(*			
	EVERDE sp. z o.o.
	Rafał Osajda		27.05.2025		TC 4024.66
	Metoda główna bazowania wywołuje metode przeciążaną Bazowanie_Cykl dziecka
*)
METHOD PRIVATE HomingCycleInternal : BOOL
VAR_INPUT
END_VAR
CASE THIS^.stHoming.cmdExecute.GetStep () OF
0	:
	IF (THIS^.stHoming.bWithoutHoming) THEN	//bazowanie wyłączone true
		THIS^.stHoming.bIsNeeded		:= TRUE;	//ustaw że juz jest wybazowane
		THIS^.stHoming.cmdExecute.SetStepAsFinal ();
	ELSE
		THIS^.stHoming.iElementHomingStep	:= 0;
		THIS^.stHoming.cmdExecute.SetStepINC10 ();
	END_IF
	THIS^.stHoming.bIsNeeded			:= TRUE;
	HomingCycleInternal				:= TRUE;
10	:
	IF (NOT THIS^.HomingCycle ()) THEN
		THIS^.stHoming.cmdExecute.SetStepAsFinal ();
	END_IF
	HomingCycleInternal				:= TRUE;
GVL_BaseConstans.FINISH_STEP	:
	THIS^.stHoming.bIsNeeded			:= FALSE;	//ustaw że juz jest wybazowane
	HomingCycleInternal				:= FALSE;
END_CASE
END_METHOD

(*			
	EVERDE sp. z o.o.
	Rafał Osajda		27.05.2025		TC 4024.66
	Bazowanie w toku
*)
METHOD PUBLIC HomingGetBusy : BOOL
VAR_INPUT
END_VAR
HomingGetBusy		:= THIS^.stHoming.cmdExecute.IsBusy ();
END_METHOD

(*			
	EVERDE sp. z o.o.
	Rafał Osajda		31.03.2025		TC 4024.66
	Flaga że w tej sesji pracy maszyny element został już wybazowany
*)
METHOD PUBLIC HomingGetDone : BOOL
VAR_INPUT
END_VAR
HomingGetDone	:= THIS^.stHoming.cmdExecute.IsDone ();
END_METHOD

(*			
	EVERDE sp. z o.o.
	Rafał Osajda		11.04.2025		TC 4024.66
	Zwraca czy bazowanie jest potrzebne
*)
METHOD PUBLIC HomingGetIsNeeded : BOOL
VAR_INPUT
END_VAR
HomingGetIsNeeded			:= THIS^.stHoming.bIsNeeded;
END_METHOD

(*			
	EVERDE sp. z o.o.
	Rafał Osajda		11.04.2025		TC 4024.66
	Ustawia czy element jest ma być bazowany czy nie
*)
METHOD PUBLIC HomingSetWithoutHoming : BOOL
VAR_INPUT
	bIN			: BOOL;
END_VAR
THIS^.stHoming.bWithoutHoming			:= bIN;
END_METHOD

(*			
	EVERDE sp. z o.o.
	Rafał Osajda		27.05.2025		TC 4024.66
	Uruchomienie metody bazowania
*)
METHOD PUBLIC HomingStart
VAR_INPUT
END_VAR
THIS^.stHoming.cmdExecute.Execute ();
END_METHOD

(*			
	EVERDE sp. z o.o.
	Rafał Osajda		30.04.2025		TC 4024.66
	Zwraca czy element jest czymś zajety
*)
METHOD PUBLIC IsDoNothing : BOOL
IsDoNothing				:= THIS^.bDoNothing;
END_METHOD

(*			
	EVERDE sp. z o.o.
	Rafał Osajda		30.04.2025		TC 4024.66
	Zwraca czy element jest w pozycji 0 - referencyjnej
*)
METHOD PUBLIC IsPosition0 : BOOL
IsPosition0				:= THIS^.bPosition0;
END_METHOD

METHOD PUBLIC IsValidCommonData : BOOL
VAR_INPUT
END_VAR

VAR
	bResult: BOOL;
	iI: INT;
END_VAR
bResult						:= SUPER^.IsValidCommonData ();

FOR iI := 1 TO TO_INT (THIS^.uiNumberOfComponents) DO
	bResult					:= bResult AND THIS^.arrComponent [iI].IsValidCommonData ();
END_FOR

IsValidCommonData			:= bResult;
END_METHOD

(*			
	EVERDE sp. z o.o.
	Rafał Osajda		07.10.2025		TC 4024.66
	Dodpisywanie się do listy logera
*)
METHOD PUBLIC JoinTheLogger : BOOL
VAR_INPUT
END_VAR

VAR
	bResult: BOOL;
	iI: INT;
END_VAR
bResult			:= SUPER^.JoinTheLogger ();

FOR iI := 1 TO  TO_INT (THIS^.uiNumberOfComponents) DO
	bResult 	:= bResult AND THIS^.arrComponent [iI].JoinTheLogger ();
END_FOR

JoinTheLogger	:= bResult;
END_METHOD

METHOD PUBLIC LinkCommonData : BOOL
VAR_INPUT
	stCommonData				: REFERENCE TO ST_BaseCommonData;
END_VAR
VAR
	bResult						: BOOL;
	iI: INT;
END_VAR
bResult							:= SUPER^.LinkCommonData (stCommonData := stCommonData);

FOR iI := 1 TO TO_INT (THIS^.uiNumberOfComponents) DO
	bResult := bResult AND THIS^.arrComponent [iI].LinkCommonData (stCommonData := stCommonData);
END_FOR

LinkCommonData					:= bResult;
END_METHOD

METHOD PUBLIC LinkSS1 : BOOL
VAR_INPUT
	fbSS1			: ITF_BaseFlagGet;
END_VAR
THIS^.itfSS1		:= fbSS1;

LinkSS1				:= THIS^.itfSS1 <> 0;
END_METHOD

METHOD PUBLIC LinkSTO : BOOL
VAR_INPUT
	fbSTO			: ITF_BaseFlagGet;
END_VAR
THIS^.itfSTO		:= fbSTO;

LinkSTO				:= THIS^.itfSTO <> 0;
END_METHOD

(*			
	EVERDE sp. z o.o.
	Rafał Osajda		31.03.2025		TC 4024.66
	Zwraca status zasilania	
*)
METHOD PUBLIC PowerGetStatus : BOOL
VAR_INPUT
END_VAR
PowerGetStatus			:= THIS^.stPower.bStatus;
END_METHOD

(*			
	EVERDE sp. z o.o.
	Rafał Osajda		13.10.2025		TC 4024.66
	Podstawowy cykl wyłączania zasilania. Dla Specyficznych urządzeń przeciążyć
*)
METHOD PROTECTED PowerOffCycle : BOOL
THIS^.stPower.bStatus		:= FALSE;
PowerOffCycle				:= FALSE;
END_METHOD

(*			
	EVERDE sp. z o.o.
	Rafał Osajda		13.10.2025		TC 4024.66
	Podstawowy cykl włączania zasilania. Dla Specyficznych urządzeń przeciążyć
*)
METHOD PROTECTED PowerOnCycle : BOOL
THIS^.stPower.bStatus		:= TRUE;
PowerOnCycle				:= FALSE;
END_METHOD

(*			
	EVERDE sp. z o.o.
	Rafał Osajda		31.03.2025		TC 4024.66
	Wyłączenie zasilania
*)
METHOD PUBLIC PowerTurnOff : BOOL
VAR_INPUT
END_VAR
THIS^.stPower.cmdTurnOff.Execute ();
END_METHOD

METHOD PUBLIC PowerTurnOffDone : BOOL
VAR_INPUT
END_VAR
PowerTurnOffDone		:= THIS^.stPower.cmdTurnOff.IsDone ();
END_METHOD

METHOD PUBLIC PowerTurnOffInProgress : BOOL
VAR_INPUT
END_VAR
PowerTurnOffInProgress			:= THIS^.stPower.cmdTurnOff.IsBusy ();
END_METHOD

(*			
	EVERDE sp. z o.o.
	Rafał Osajda		31.03.2025		TC 4024.66
	Uruchomienie zasialania
*)
METHOD PUBLIC PowerTurnOn
VAR_INPUT
END_VAR
THIS^.stPower.cmdTurnOn.Execute ();
END_METHOD

METHOD PUBLIC PowerTurnOnDone : BOOL
VAR_INPUT
END_VAR
PowerTurnOnDone		:= THIS^.stPower.cmdTurnOn.IsDone ();
END_METHOD

METHOD PUBLIC PowerTurnOnInProgress : BOOL
VAR_INPUT
END_VAR
PowerTurnOnInProgress		:= THIS^.stPower.cmdTurnOn.IsBusy ();
END_METHOD

METHOD PROTECTED ResetOperation : BOOL
VAR
	bResult				: BOOL;
END_VAR
bResult					:= SUPER^.ResetOperation ();

THIS^.stHoming.bIsNeeded	:= TRUE;
THIS^.stHoming.cmdExecute.Abort ();
THIS^.stHoming.iChildHomingStep	:= 0;
THIS^.stHoming.iElementHomingStep	:= 0;

ResetOperation			:= FALSE OR bResult;
END_METHOD

METHOD PUBLIC SetCode
VAR_INPUT
	sCode							: STRING;
	sAdd							: STRING;
END_VAR
VAR
	sItemCode						: STRING;
	iI								: INT;
	sComponentCode					: STRING;
END_VAR
sItemCode		:=  CreateElementCode (sParentCode := sCode, sAdd := sAdd);
SUPER^.SetCode (sCode := sItemCode, sAdd := '');

FOR iI := 1 TO TO_INT (THIS^.uiNumberOfComponents) DO
	sComponentCode	:= CreateElementCode (sParentCode := sItemCode, sAdd := TO_STRING (iI));
	THIS^.arrComponent [iI].SetCode (sCode	:= sComponentCode, sAdd := '');
END_FOR
END_METHOD

(*			
	EVERDE sp. z o.o.
	Rafał Osajda		03.10.2025		TC 4024.66
	nadawanie unikalnych ID dla zdarzeń
*)
METHOD PUBLIC SetEventsIDs : UINT
VAR_INPUT
	uiNewID		: UINT;
END_VAR
VAR
	iI			: INT;
	uiLastID	: UINT;
END_VAR
uiLastID		:= SUPER^.SetEventsIDs (uiNewID	:= uiNewID);

FOR iI := 1 TO TO_INT (THIS^.uiNumberOfComponents) DO 
	uiLastID			:= THIS^.arrComponent [iI].SetEventsIDs (uiNewID	:= uiLastID);
END_FOR
SetEventsIDs				:= uiLastID;
END_METHOD

METHOD PUBLIC SetID : UINT
VAR_INPUT
	uiID					: UINT;
END_VAR
VAR
	uiLastID				: UINT;
	iI						: INT;
END_VAR
uiLastID				:= SUPER^.SetID (uiID	:= uiID);

FOR iI := 1 TO TO_INT (THIS^.uiNumberOfComponents) DO 
	uiLastID			:= THIS^.arrComponent [iI].SetID (uiID	:= uiLastID + 1);
END_FOR
SetID					:= uiLastID;
END_METHOD

END_FUNCTION_BLOCK

// ---- POUs/A06_FB_BaseGroupElement/FB_BaseGroupElement.TcPOU
(*			
	RAFALOS
	Rafał Osajda		19.09.2025		TC 4024.66
	FB Bazowy dla wszystkich elementów złożonych
*)
FUNCTION_BLOCK FB_BaseGroupElement EXTENDS FB_BaseControlElement IMPLEMENTS ITF_BaseGroupElement, ITF_BaseGroupElement_HMI_Connector, ITF_BaseMessengerRecipient, ITF_BaseMessengerSender
VAR
	arrControlElement			: ARRAY [1..GVL_BaseConstans.MAX_ITEM_PER_ELEMENT] OF ITF_BaseControlElement;
	uiNumberOfControlElement	: UINT;
	itfCommunicator				: ITF_BaseCommunicator;
END_VAR

METHOD PROTECTED AddControlElement : BOOL
VAR_INPUT
	itfControlElement		: ITF_BaseControlElement;
END_VAR
IF (THIS^.uiNumberOfControlElement + 1 <= GVL_BaseConstans.MAX_ITEM_PER_ELEMENT) THEN
	THIS^.uiNumberOfControlElement		:= THIS^.uiNumberOfControlElement + 1;
	THIS^.arrControlElement [THIS^.uiNumberOfControlElement]	:= itfControlElement;
	AddControlElement			:= TRUE;
ELSE
	;//zwrocenie zbyt dużo komponentow
END_IF
END_METHOD

METHOD PUBLIC ConfirmReceipt : BOOL
VAR_INPUT
	sText: STRING;
END_VAR
ConfirmReceipt	:= THIS^.itfCommunicator.ReceiveDataConfirm (sText := sText, itfRecipient := THIS^);
END_METHOD

(*			
	RafalOS
	Rafał Osajda		27.03.2025		TC 4024.66
	Obsluga bledow sprawdzanie czy jakis blad sie nei pojawil i ustawienie stanu lub wylaczenie
*)
METHOD PUBLIC ExecuteEveryCycle_Error
VAR
	iI					: INT;
END_VAR
SUPER^.ExecuteEveryCycle_Error ();

FOR iI := 1 TO TO_INT (THIS^.uiNumberOfControlElement) DO
	THIS^.arrControlElement [iI].ExecuteEveryCycle_Error ();
END_FOR
END_METHOD

(*			
	RafalOS
	Rafał Osajda		27.03.2025		TC 4024.66
	Wywolanie co cykl operacji 
*)
METHOD PUBLIC ExecuteEveryCycle_Operation
VAR
	iI				: INT;
END_VAR
SUPER^.ExecuteEveryCycle_Operation ();

FOR iI := 1 TO TO_INT (THIS^.uiNumberOfControlElement) DO
	THIS^.arrControlElement [iI].ExecuteEveryCycle_Operation ();
END_FOR
END_METHOD

(*			
	RafalOS
	Rafał Osajda		27.03.2025		TC 4024.66
	Aktualizacja flag 
*)
METHOD PUBLIC ExecuteEveryCycle_Status
VAR
	iI				: INT;
END_VAR
SUPER^.ExecuteEveryCycle_Status ();

FOR iI := 1 TO TO_INT (THIS^.uiNumberOfControlElement) DO
	THIS^.arrControlElement [iI].ExecuteEveryCycle_Status ();
END_FOR
END_METHOD

(*			
	RafalOS
	Rafał Osajda		27.03.2025		TC 4024.66
	Testowanie czy nei pojawil sie jakis rozkaz i uruchomienie odpowiednich operacji
*)
METHOD PUBLIC ExecuteEveryCycle_Test
VAR
	iI			: INT;
END_VAR
SUPER^.ExecuteEveryCycle_Test ();

FOR iI := 1 TO TO_INT (THIS^.uiNumberOfControlElement) DO
	THIS^.arrControlElement [iI].ExecuteEveryCycle_Test ();
END_FOR
END_METHOD

METHOD FB_init : BOOL
VAR_INPUT
	bInitRetains : BOOL; // if TRUE, the retain variables are initialized (warm start / cold start)
	bInCopyCode : BOOL;  // if TRUE, the instance afterwards gets moved into the copy code (online change)
END_VAR
THIS^.stIdentifier.eType			:= E_BaseElementType.eGroup;
END_METHOD

METHOD PUBLIC FirstCycle : BOOL
VAR_INPUT
END_VAR
VAR
	bResult			: bool;
	iI				: INT;
END_VAR
bResult				:= SUPER^.FirstCycle ();

FOR iI := 1 TO TO_INT (THIS^.uiNumberOfControlElement) DO
	bResult			:= bResult AND THIS^.arrControlElement [iI].FirstCycle ();
END_FOR

FirstCycle			:= bResult;
END_METHOD

METHOD GetITFGroupElement : ITF_BaseGroupElement
VAR_INPUT
END_VAR
GetITFGroupElement	:= THIS^;
END_METHOD

METHOD GetITFTopElement : ITF_BaseTopElement
VAR_INPUT
END_VAR
GetITFTopElement		:= null;
END_METHOD

(*			
	RafalOS
	Rafał Osajda		27.05.2025		TC 4024.66
	Metoda bazowania kontrektnego elementu 
*)
METHOD PROTECTED HomingCycle : BOOL
VAR
	iI			: INT;
END_VAR
CASE THIS^.stHoming.iElementHomingStep OF
0	:
	FOR iI := 1 TO TO_INT (THIS^.uiNumberOfControlElement) DO
		THIS^.arrControlElement [iI].HomingStart ();
	END_FOR
	THIS^.stHoming.iElementHomingStep	:= THIS^.stHoming.iElementHomingStep + 10;
	HomingCycle							:= TRUE;
10	:
	THIS^.stHoming.iElementHomingStep	:= THIS^.stHoming.iElementHomingStep + 10;
	HomingCycle							:= TRUE;
20	:
	IF (THIS^.HomingGetDone ()) THEN
		THIS^.stHoming.iElementHomingStep 	:= GVL_BaseConstans.FINISH_STEP;
	END_IF	
	HomingCycle							:= TRUE;
GVL_BaseConstans.FINISH_STEP :
	HomingCycle							:= FALSE;
END_CASE
END_METHOD

(*			
	RafalOS
	Rafał Osajda		31.03.2025		TC 4024.66
	Flaga że w tej sesji pracy maszyny element został już wybazowany
*)
METHOD PUBLIC HomingGetDone : BOOL
VAR
	iI				: INT;
	btmpHomingDone	: BOOL;
END_VAR
btmpHomingDone		:= TRUE;
FOR iI := 1 TO TO_INT (THIS^.uiNumberOfControlElement) DO
	btmpHomingDone	:= btmpHomingDone AND THIS^.arrControlElement [iI].HomingGetDone ();
	IF (NOT btmpHomingDone) THEN
		EXIT;
	END_IF
END_FOR
HomingGetDone		:= btmpHomingDone;
END_METHOD

(*			
	RafalOS
	Rafał Osajda		11.04.2025		TC 4024.66
	Zwraca czy bazowanie jest potrzebne
*)
METHOD PUBLIC HomingGetIsNeeded : BOOL
VAR
	btmpHomingIsNeeded	: BOOL := FALSE;
	iI					: INT;
END_VAR
FOR iI := 1 TO TO_INT (THIS^.uiNumberOfControlElement) DO
	btmpHomingIsNeeded	:= btmpHomingIsNeeded OR THIS^.arrControlElement [iI].HomingGetIsNeeded ();
	IF (btmpHomingIsNeeded) THEN
		EXIT;
	END_IF
END_FOR
HomingGetIsNeeded		:= btmpHomingIsNeeded;
END_METHOD

(*			
	RafalOS
	Rafał Osajda		30.04.2025		TC 4024.66
	Zwraca czy element jest czymś zajety
*)
METHOD PUBLIC IsDoNothing : BOOL
VAR
	iI				: INT;
	btmpDoNothing	: BOOL := TRUE;
END_VAR
FOR iI := 1 TO TO_INT (THIS^.uiNumberOfControlElement) DO
	btmpDoNothing		:= btmpDoNothing AND THIS^.arrControlElement [iI].IsDoNothing ();
	IF (NOT btmpDoNothing) THEN
		EXIT;
	END_IF
END_FOR
THIS^.bDoNothing		:= btmpDoNothing;
IsDoNothing			:= btmpDoNothing;
END_METHOD

(*			
	RafalOS
	Rafał Osajda		30.04.2025		TC 4024.66
	Zwraca czy element jest w pozycji 0 - referencyjnej
*)
METHOD PUBLIC IsPosition0 : BOOL
VAR
	iI					: INT;
	btmpPosition0		: BOOL;
END_VAR
FOR iI := 1 TO TO_INT (THIS^.uiNumberOfControlElement) DO
	btmpPosition0		:= btmpPosition0 AND THIS^.arrControlElement [iI].IsPosition0 ();
	IF (NOT btmpPosition0) THEN
		EXIT;
	END_IF
END_FOR
THIS^.bPosition0		:= btmpPosition0;
IsPosition0			:= btmpPosition0;
END_METHOD

METHOD PUBLIC IsValidCommonData : BOOL
VAR_INPUT
END_VAR

VAR
	bResult: BOOL;
	iI: INT;
END_VAR
bResult						:= SUPER^.IsValidCommonData ();

FOR iI := 1 TO TO_INT (THIS^.uiNumberOfControlElement) DO
	bResult					:= bResult AND THIS^.arrControlElement [iI].IsValidCommonData ();
END_FOR

IsValidCommonData			:= bResult;
END_METHOD

(*			
	RafalOS
	Rafał Osajda		07.10.2025		TC 4024.66
	Dodpisywanie się do listy logera
*)
METHOD PUBLIC JoinTheLogger : BOOL
VAR_INPUT
END_VAR

VAR
	bResult: BOOL;
	iI: INT;
END_VAR
bResult			:= SUPER^.JoinTheLogger ();

FOR iI := 1 TO  TO_INT (THIS^.uiNumberOfControlElement) DO
	bResult 	:= bResult AND THIS^.arrControlElement [iI].JoinTheLogger ();
END_FOR

JoinTheLogger	:= bResult;
END_METHOD

METHOD PUBLIC LinkCommonData : BOOL
VAR_INPUT
	stCommonData				: REFERENCE TO ST_BaseCommonData;
END_VAR
VAR
	bResult						: BOOL;
	iI: INT;
END_VAR
bResult							:= SUPER^.LinkCommonData (stCommonData := stCommonData);

FOR iI := 1 TO TO_INT (THIS^.uiNumberOfControlElement) DO
	bResult := bResult AND THIS^.arrControlElement [iI].LinkCommonData (stCommonData := stCommonData);
END_FOR

LinkCommonData					:= bResult;
END_METHOD

METHOD PUBLIC LinkCommunicator : BOOL
VAR_INPUT
	fbCommunicator				: ITF_BaseCommunicator;
END_VAR
THIS^.itfCommunicator			:= fbCommunicator;
IF (THIS^.itfCommunicator <> 0) THEN
	LinkCommunicator			:= TRUE;
END_IF
END_METHOD

METHOD PUBLIC LinkSS1 : BOOL
VAR_INPUT
	fbSS1			: ITF_BaseFlagGet;
END_VAR

VAR
	bresult: BOOL;
	iI: INT;
END_VAR
bresult				:= SUPER^.LinkSS1 (fbSS1 := fbSS1);

FOR iI := 1 TO TO_INT (THIS^.uiNumberOfControlElement) DO
	bresult			:= bresult AND THIS^.arrControlElement [iI].LinkSS1 (fbSS1	:= fbSS1);
END_FOR

LinkSS1				:= bresult;
END_METHOD

METHOD PUBLIC LinkSTO : BOOL
VAR_INPUT
	fbSTO			: ITF_BaseFlagGet;
END_VAR

VAR
	bresult: BOOL;
	iI: INT;
END_VAR
bresult				:= SUPER^.LinkSTO (fbSTO := fbSTO);

FOR iI := 1 TO TO_INT (THIS^.uiNumberOfControlElement) DO
	bresult			:= bresult AND THIS^.arrControlElement [iI].LinkSTO (fbSTO	:= fbSTO);
END_FOR

LinkSTO				:= bresult;
END_METHOD

METHOD PROTECTED PowerOffCycle : BOOL
VAR
	iI							: INT;
	bPowerStatus			: BOOL;
END_VAR
CASE stPower.cmdTurnOff.GetStep () OF
0	:
	FOR iI := 1 TO TO_INT (THIS^.uiNumberOfControlElement) DO
		THIS^.arrControlElement [iI].PowerTurnOff ();
	END_FOR
	THIS^.stPower.cmdTurnOff.SetStepINC10 ();
	PowerOffCycle			:= TRUE;
10	:
	bPowerStatus			:= FALSE;
	FOR iI := 1 TO TO_INT (THIS^.uiNumberOfControlElement) DO
		bPowerStatus		:= bPowerStatus OR THIS^.arrControlElement [iI].PowerGetStatus ();
		IF (bPowerStatus) THEN
			EXIT;
		END_IF
	END_FOR	
	IF (NOT bPowerStatus) THEN
		THIS^.stPower.bStatus	:= FALSE;
		THIS^.stPower.cmdTurnOff.SetStepAsFinal ();
	ELSE
		PowerOffCycle			:= TRUE;
	END_IF	
END_CASE
END_METHOD

METHOD PROTECTED PowerOnCycle : BOOL
VAR
	iI						: INT;
	bPowerStatus		: BOOL;
END_VAR
CASE stPower.cmdTurnOn.GetStep () OF
0	:
	FOR iI := 1 TO TO_INT (THIS^.uiNumberOfControlElement) DO
		THIS^.arrControlElement [iI].PowerTurnOn ();
	END_FOR
	THIS^.stPower.cmdTurnOn.SetStepINC10 ();
	PowerOnCycle				:= TRUE;
10	:
	bPowerStatus			:= TRUE;
	FOR iI := 1 TO TO_INT (THIS^.uiNumberOfControlElement) DO
		bPowerStatus		:= bPowerStatus AND THIS^.arrControlElement [iI].PowerGetStatus ();
		IF (NOT bPowerStatus) THEN
			EXIT;
		END_IF
	END_FOR	
	IF (bPowerStatus) THEN
		THIS^.stPower.bStatus	:= TRUE;
		THIS^.stPower.cmdTurnOn.SetStepAsFinal ();
		PowerOnCycle			:= FALSE;
	ELSE
		PowerOnCycle			:= TRUE;
	END_IF	
END_CASE
END_METHOD

METHOD PUBLIC Receive_BOOL : BOOL
VAR_INPUT
	sText		: STRING;
END_VAR
VAR_OUTPUT
	bValue		: BOOL;	
END_VAR
Receive_BOOL			:= THIS^.itfCommunicator.ReceiveData_BOOL (sText := sText, itfRecipient := THIS^, bValue => bValue);
END_METHOD

METHOD PUBLIC Receive_REAL : BOOL
VAR_INPUT
	sText		: STRING;
END_VAR
VAR_OUTPUT
	rValue		: REAL;	
END_VAR
Receive_REAL			:=  THIS^.itfCommunicator.ReceiveData_REAL (sText := sText, itfRecipient := THIS^, rValue => rValue);
END_METHOD

METHOD PROTECTED ResetOperation : BOOL
VAR
	bResult				: BOOL;
END_VAR
bResult					:= SUPER^.ResetOperation ();


ResetOperation			:= FALSE OR bResult;
END_METHOD

METHOD Send_BOOL : BOOL
VAR_INPUT
	sText				: STRING;
END_VAR
Send_BOOL		:= THIS^.itfCommunicator.SendData_BOOL (sText := sText, itfSender := THIS^);
END_METHOD

METHOD Send_REAL : BOOL
VAR_INPUT
	sText		: STRING;
	rValue		: REAL;
END_VAR
Send_REAL			:= THIS^.itfCommunicator.SendData_REAL (sText := sText, rValue := rValue, itfSender := THIS^);
END_METHOD

METHOD PUBLIC SetCode
VAR_INPUT
	sCode							: STRING;
	sAdd							: STRING;
END_VAR
VAR
	sItemCode						: STRING;
	iI								: INT;
	sParentCode						: STRING;
	arrSegment						: ARRAY [0..GVL_BaseConstans.MAX_NESTING_LEVEL] OF STRING;
	iDotPosition					: INT;
	iLast							: INT;
	
END_VAR
//sKodRodzica	:=  UtworzKodElementu (sKodRodzica := sKod, sDopisz := TO_STRING (THIS^.zwrocID ()));
SUPER^.SetCode (sCode := sCode, sAdd := sAdd);
sParentCode						:= THIS^.GetCode ();

IF (THIS^.uiNumberOfComponents > 0) THEN
	arrSegment [0]				:= THIS^.arrComponent [THIS^.uiNumberOfComponents].GetCode ();
	FOR iI := 1 TO TO_INT (GVL_BaseConstans.MAX_NESTING_LEVEL) DO
		iDotPosition			:= find (STR1 := arrSegment [0], STR2 := '.');
		IF (iDotPosition = 0) THEN
			arrSegment [iI]	:= arrSegment [0];
			EXIT;
		ELSE
			arrSegment [iI]		:= Tc2_Standard.LEFT (STR := arrSegment [0], SIZE := iDotPosition - 1);
			arrSegment [0]		:= Tc2_Standard.DELETE (STR := arrSegment [0], POS := 1, LEN := iDotPosition);
		END_IF
	END_FOR
	FOR iI := 0 TO TO_INT (GVL_BaseConstans.MAX_NESTING_LEVEL) - 1 DO
		IF (TO_INT (arrSegment [TO_INT (GVL_BaseConstans.MAX_NESTING_LEVEL) - iI]) <> 0 ) THEN
			iLast			:= TO_INT (arrSegment [TO_INT (GVL_BaseConstans.MAX_NESTING_LEVEL) - iI]);
			EXIT;
		END_IF
	END_FOR
END_IF

FOR iI := 1 TO TO_INT (THIS^.uiNumberOfControlElement) DO
//	sKodKomponentu	:= UtworzKodElementu (sKodRodzica := sKod, sDopisz := TO_STRING (iI));
	THIS^.arrControlElement [iI].SetCode (sCode	:= sParentCode, sAdd := TO_STRING (iI + iLast));
END_FOR
END_METHOD

(*			
	RafalOS
	Rafał Osajda		03.10.2025		TC 4024.66
	nadawanie unikalnych ID dla zdarzeń
*)
METHOD PUBLIC SetEventsIDs : UINT
VAR_INPUT
	uiNewID		: UINT;
END_VAR
VAR
	iI			: INT;
	uiLastID	: UINT;
END_VAR
uiLastID		:= SUPER^.SetEventsIDs (uiNewID	:= uiNewID);

FOR iI := 1 TO TO_INT (THIS^.uiNumberOfControlElement) DO 
	uiLastID			:= THIS^.arrControlElement [iI].SetEventsIDs (uiNewID	:= uiLastID);
END_FOR
SetEventsIDs				:= uiLastID;
END_METHOD

METHOD PUBLIC SetID : UINT
VAR_INPUT
	uiID					: UINT;
END_VAR
VAR
	uiLastID				: UINT;
	iI						: INT;
END_VAR
uiLastID				:= SUPER^.SetID (uiID	:= uiID);

FOR iI := 1 TO TO_INT (THIS^.uiNumberOfControlElement) DO 
	uiLastID			:= THIS^.arrControlElement [iI].SetID (uiID	:= uiLastID + 1);
END_FOR
SetID					:= uiLastID;
END_METHOD

END_FUNCTION_BLOCK

// ---- POUs/A07_FB_BaseTopElement/FB_BaseTopElement.TcPOU
(*			
	RAFALOS
	Rafał Osajda		19.09.2025		TC 4024.66
	Rodzic dla wszystkich podzespołów głównych w maszynie 
*)
FUNCTION_BLOCK FB_BaseTopElement EXTENDS FB_BaseGroupElement IMPLEMENTS ITF_BaseTopElement, ITF_BaseTopElement_HMI_Connector
VAR
	refstRecipe				: REFERENCE TO ST_BaseRecipe;	//referencja do wybranej receptury
	itfSaM					: ITF_BaseSaM;
END_VAR

(*			
	RafalOS
	Rafał Osajda		27.03.2025		TC 4024.66
	Obsluga bledow sprawdzanie czy jakis blad sie nei pojawil i ustawienie stanu lub wylaczenie
*)
METHOD PUBLIC ExecuteEveryCycle_Error
VAR_INPUT
END_VAR
SUPER^.ExecuteEveryCycle_Error ();
END_METHOD

(*			
	RafalOS
	Rafał Osajda		27.03.2025		TC 4024.66
	Wywolanie co cykl operacji 
*)
METHOD PUBLIC ExecuteEveryCycle_Operation
VAR_INPUT
END_VAR
SUPER^.ExecuteEveryCycle_Operation ();
END_METHOD

(*			
	RafalOS
	Rafał Osajda		27.03.2025		TC 4024.66
	Aktualizacja flag 
*)
METHOD PUBLIC ExecuteEveryCycle_Status
VAR_INST
END_VAR
SUPER^.ExecuteEveryCycle_Status ();
END_METHOD

(*			
	RafalOS
	Rafał Osajda		27.03.2025		TC 4024.66
	Testowanie czy nei pojawil sie jakis rozkaz i uruchomienie odpowiednich operacji
*)
METHOD PUBLIC ExecuteEveryCycle_Test
VAR_INPUT
END_VAR
SUPER^.ExecuteEveryCycle_Test ();
END_METHOD

METHOD FB_init : BOOL
VAR_INPUT
	bInitRetains : BOOL; // if TRUE, the retain variables are initialized (warm start / cold start)
	bInCopyCode : BOOL;  // if TRUE, the instance afterwards gets moved into the copy code (online change)
END_VAR
THIS^.stIdentifier.eType			:= E_BaseElementType.eTop;
END_METHOD

METHOD GetITFTopElement : ITF_BaseTopElement
VAR_INPUT
END_VAR
GetITFTopElement		:= THIS^;
END_METHOD

METHOD PUBLIC IsValidLinkSAM : BOOL
IsValidLinkSAM	:= THIS^.itfSAM <> 0;
END_METHOD

METHOD PUBLIC LinkSAM : BOOL
VAR_INPUT
	fbSAM				: ITF_BaseSAM;
END_VAR
THIS^.itfSAM			:= fbSAM;
END_METHOD

(*			RafalOS
	Rafał Osajda		27.10.2024		TC 4026.11		wer. 0.0.0.1
	metoda obsługi czekania na reset
*)
METHOD SP_Aborted : BOOL
END_METHOD

(*			RafalOS
	Rafał Osajda		27.10.2024		TC 4026.11		wer. 0.0.0.1
	metoda obsługi wyłączania napędów po wciśnięciu grzyba
*)
METHOD SP_Aborting : BOOL
IF (NOT THIS^.itfSAM.IsChangeModeBusy ()) THEN
	IF (THIS^.stPower.bStatus AND NOT THIS^.stPower.cmdTurnOff.IsBusy ()) THEN
		THIS^.stPower.cmdTurnOff.Execute ();
	END_IF
	IF (NOT THIS^.stPower.bStatus AND THIS^.stPower.cmdTurnOff.IsDone ()) THEN
		SP_Aborting								:= TRUE;
		THIS^.Reset ();
	ELSE
		SP_Aborting								:= FALSE;
	END_IF
END_IF
END_METHOD

(*			RafalOS
	Rafał Osajda		27.10.2024		TC 4026.11		wer. 0.0.0.1
	metoda obsługi czyszczenia po grzybie
*)
METHOD SP_Clearing : BOOL
IF (NOT THIS^.stPower.bStatus AND NOT THIS^.stPower.cmdTurnOn.IsBusy ()
	AND THIS^.itfSS1.GetFlag () AND THIS^.itfSTO.GetFlag ()) THEN
	THIS^.stPower.cmdTurnOn.Execute ();
END_IF
IF (THIS^.stPower.bStatus AND THIS^.stPower.cmdTurnOn.IsDone ()) THEN
	SP_Clearing								:= TRUE;
ELSE
	SP_Clearing								:= FALSE;
END_IF
END_METHOD

(*			RafalOS
	Rafał Osajda		27.10.2024		TC 4026.11		wer. 0.0.0.1
	metoda obsługi Wykonania określonego zadania
*)
METHOD SP_Complete : BOOL
END_METHOD

(*			RafalOS
	Rafał Osajda		27.10.2024		TC 4026.11		wer. 0.0.0.1
	metoda obsługi pracy automatycznej do zadanej wartości ilości elementów
*)
METHOD SP_Completing : BOOL
SP_Completing				:= TRUE;
END_METHOD

(*			RafalOS
	Rafał Osajda		27.10.2024		TC 4026.11		wer. 0.0.0.1
	metoda obsługi pracy
*)
METHOD SP_Execute : BOOL
CASE THIS^.itfSAM.GetMode () OF
	E_BaseMachineMode.NotAllowed	    : ;	
	E_BaseMachineMode.Production		: SP_Execute_1_Production ();
	E_BaseMachineMode.Maintenance		: SP_Execute_2_Maintenance ();
	E_BaseMachineMode.Manual			: SP_Execute_3_Manual ();
	E_BaseMachineMode.Washing			: SP_Execute_4_Washing ();
	E_BaseMachineMode.Diagnostics		: SP_Execute_5_Diagnostics ();
//	E_TrybyPracy.Uzytkownika2			: SP_Execute_6_Uzytkownika2 ();
//	E_TrybyPracy.Uzytkownika3			: SP_Execute_7_Uzytkownika3 ();
//	E_TrybyPracy.Uzytkownika4			: SP_Execute_8_Uzytkownika4 ();
//	E_TrybyPracy.Uzytkownika5			: SP_Execute_9_Uzytkownika5 ();
END_CASE
END_METHOD

(*			RafalOS
	Rafał Osajda		27.10.2024		TC 4026.11		wer. 0.0.0.1
	metoda obsługi pracy
*)
METHOD PROTECTED SP_Execute_1_Production : BOOL
VAR_INPUT
//	eTrybPracy								: OTP.E_TrybyPracy;
END_VAR
END_METHOD

(*			RafalOS
	Rafał Osajda		27.10.2024		TC 4026.11		wer. 0.0.0.1
	metoda obsługi pracy
*)
METHOD SP_Execute_2_Maintenance : BOOL
VAR_INPUT
//	eTrybPracy								: OTP.E_TrybyPracy;
END_VAR
END_METHOD

(*			RafalOS
	Rafał Osajda		27.10.2024		TC 4026.11		wer. 0.0.0.1
	metoda obsługi pracy
*)
METHOD SP_Execute_3_Manual : BOOL
VAR_INPUT
//	eTrybPracy								: OTP.E_TrybyPracy;
END_VAR
END_METHOD

(*			RafalOS
	Rafał Osajda		27.10.2024		TC 4026.11		wer. 0.0.0.1
	metoda obsługi pracy
*)
METHOD SP_Execute_4_Washing : BOOL
VAR_INPUT
//	eTrybPracy								: OTP.E_TrybyPracy;
END_VAR
END_METHOD

(*			RafalOS
	Rafał Osajda		27.10.2024		TC 4026.11		wer. 0.0.0.1
	metoda obsługi pracy
*)
METHOD SP_Execute_5_Diagnostics : BOOL
VAR_INPUT
//	eTrybPracy								: OTP.E_TrybyPracy;
END_VAR
END_METHOD

(*			RafalOS
	Rafał Osajda		27.10.2024		TC 4026.11		wer. 0.0.0.1
	metoda obsługi wstrzymania pracy ze względów na błędy/alarmy
*)
METHOD SP_Held : BOOL
END_METHOD

(*			RafalOS
	Rafał Osajda		27.10.2024		TC 4026.11		wer. 0.0.0.1
	metoda obsługi wyjścia z wstrzymania pracy
*)
METHOD SP_Holding : BOOL
//wstrzymywanie pracy ze wzgledu na okoliczności wewnetrzne
SP_Holding									:= TRUE;
END_METHOD

(*			RafalOS
	Rafał Osajda		27.10.2024		TC 4026.11		wer. 0.0.0.1
	metoda obsługi czekania na dalsze rozkazy
*)
METHOD SP_Idle : BOOL
END_METHOD

(*			RafalOS
	Rafał Osajda		27.10.2024		TC 4026.11		wer. 0.0.0.1
	Metoda sprawdzająca czy elementy maszyny ustawiły się na 0 wczytanie parametrów pracy
*)
METHOD SP_Resetting : BOOL
IF (NOT THIS^.stHoming.bIsNeeded OR THIS^.itfSAM.GetMode () = E_BaseMachineMode.Maintenance) THEN
	SP_Resetting				:= TRUE;
ELSE
	IF (NOT THIS^.stHoming.cmdExecute.IsBusy ()) THEN
		THIS^.stHoming.cmdExecute.Execute ();
	END_IF
	SP_Resetting				:= FALSE;
END_IF
END_METHOD

(*			RafalOS
	Rafał Osajda		27.10.2024		TC 4026.11		wer. 0.0.0.1
	metoda obsługi uruchamiania pracy
*)
METHOD SP_Starting : BOOL
(* w razie potrzeby tutaj ustawiać flagi przy starcie pracy maszyny *)
//uruchamianie cykli maszyny
SP_Starting									:= TRUE;
END_METHOD

(*			RafalOS
	Rafał Osajda		27.10.2024		TC 4026.11		wer. 0.0.0.1
	metoda obsługi czekania na dalsze rozkazy
*)
METHOD SP_Stopped : BOOL
END_METHOD

(*			RafalOS
	Rafał Osajda		27.10.2024		TC 4026.11		wer. 0.0.0.1
	Metoda sprawdzająca czy wszystkie operacje zostały już zakończone i można wyłaczyc pracę 
*)
METHOD SP_Stopping : BOOL
IF (THIS^.IsDoNothing ()) THEN	//nic nie robi
	SP_Stopping					:= TRUE;
ELSE
//	SUPER^.BazowanieWylacz ();
	SP_Stopping					:= FALSE;
END_IF
END_METHOD

(*			RafalOS
	Rafał Osajda		27.10.2024		TC 4026.11		wer. 0.0.0.1
	metoda obsługi wstrzymania pracy ze względu na warunki zewnętrzne np brak materialu
*)
METHOD SP_Suspended : BOOL
END_METHOD

(*			RafalOS
	Rafał Osajda		27.10.2024		TC 4026.11		wer. 0.0.0.1
	metoda obsługi zawieszania pracy ze wzgledu na okoliczności zewnętrzne
*)
METHOD SP_Suspending : BOOL
//zawieszanie pracy ne względu na okoliczności zewnętrzne
SP_Suspending								:= TRUE;
END_METHOD

(*			RafalOS
	Rafał Osajda		27.10.2024		TC 4026.11		wer. 0.0.0.1
	metoda obsługi stanu zabroniownego - występuje tylko przy starcie
*)
METHOD SP_Undefined : BOOL
END_METHOD

(*			RafalOS
	Rafał Osajda		27.10.2024		TC 4026.11		wer. 0.0.0.1
	metoda obsługi uruchamiania po wstrzymaniu
*)
METHOD SP_Unholding : BOOL
//warunek wyjścia z stanu wstzrymania pracy
SP_Unholding								:= TRUE;
END_METHOD

(*			RafalOS
	Rafał Osajda		27.10.2024		TC 4026.11		wer. 0.0.0.1
	metoda obsługi uruchamiania po wstzryamaniu
*)
METHOD SP_Unsuspending : BOOL
//warunek wyjścia z stanu wstzrymania pracy
SP_Unsuspending							:= TRUE;
END_METHOD

END_FUNCTION_BLOCK

// ---- POUs/B02_Recipes/FB_BaseRecipe.TcPOU
(*			
	RafalOS
	Rafał Osajda		28.02.2025		TC 4026.13		wer. 0.0.0.1
	Obsługa receptur
*)
FUNCTION_BLOCK FB_BaseRecipe EXTENDS FB_Base IMPLEMENTS ITF_BaseCreatingTemplateMethod
VAR
	bChoose						: BOOL;		//receptura wybrana
	iNumberToChoose				: INT;		//numer wybranej
	arritfCreatingRecipe		: ARRAY [1..GVL_BaseConstans.MAX_NUMBER_OF_TEMPLATES] OF ITF_BaseCreateTemplateOfRecipe;
	uiNumberOfCreatingRecipe	: UINT;		//ilosc fb dla tworzenia receptur
END_VAR
VAR PERSISTENT
	arrTemplates				: ARRAY [1..GVL_BaseConstans.MAX_NUMBER_OF_TEMPLATES] OF ST_BaseRecipe;	//szablony
	arrRecipes					: ARRAY [1..GVL_BaseConstans.MAX_NUMBER_OF_RECIPES] OF ST_BaseRecipe;	//receptury
	uiNumberOfTemplates			: UINT;			//ilość dodanych szablonów
	uiNumberOfRecipes			: UINT;			//ilość dodanych receptur
	uiChosen					: UINT;			//numer wybranej receptruy		
	stChosen					: ST_BaseRecipe;	//kopia wybranej recepury kopiowana w momencie wyboru, zmiany w recepturze bazowej nie jest przepisywana automatycznia
END_VAR

(*			
	RafalOS
	Rafał Osajda		25.10.2025		TC 4024.66
	Dodawanie składnika do szablonu
*)
METHOD PUBLIC AddIngredientToTemplate : BOOL
VAR_INPUT
	uiNumber		: UINT;
	stIngredient	: ST_BaseDescriptor;
END_VAR
IF (THIS^.arrTemplates [uiNumber].uiNumber + 1 <= GVL_BaseConstans.MAX_NUMBER_Of_INGREDIENTS) THEN
	THIS^.arrTemplates [uiNumber].uiNumber			:= THIS^.arrTemplates [uiNumber].uiNumber + 1;
	THIS^.arrTemplates [uiNumber].arrIngredient [THIS^.arrTemplates [uiNumber].uiNumber]	:= stIngredient;
//	THIS^.arrSzablony [uiNumer].arrSkladnik [THIS^.arrSzablony [uiNumer].uiIlosc].PowiarzJezyk (fbLokalizacja := THIS^.itfJezyk);
	AddIngredientToTemplate						:= TRUE;
END_IF
END_METHOD

(*			
	RafalOS
	Rafał Osajda		25.10.2025		TC 4024.66
	Dodanie itferfejsu FB dla tworzenia szablonów receptur z programu maszyny
*)
METHOD PUBLIC AddITFToCreateTemplate : BOOL
VAR_INPUT
	fbToCtreateTemplate		: ITF_BaseCreateTemplateOfRecipe;
END_VAR
IF (THIS^.uiNumberOfCreatingRecipe + 1 <= GVL_BaseConstans.MAX_NUMBER_OF_TEMPLATES) THEN
	THIS^.uiNumberOfCreatingRecipe	:= THIS^.uiNumberOfCreatingRecipe + 1;
	THIS^.arritfCreatingRecipe [THIS^.uiNumberOfCreatingRecipe]	:= fbToCtreateTemplate;
	AddITFToCreateTemplate		:= TRUE;
ELSE
	AddITFToCreateTemplate		:= FALSE;
END_IF
END_METHOD

(*			
	RafalOS
	Rafał Osajda		03.03.2025		TC 4026.13		wer. 0.0.0.1
	Kopiuje składniki z wybranej receptury i tworzy nową recepture
*)
METHOD PUBLIC AddRecipeFromRecipe : BOOL
VAR_INPUT
	uiNumberRecipe				: UINT;
	stTexts						: ST_BaseLabel;
END_VAR
IF (THIS^.uiNumberOfRecipes + 1 <= GVL_BaseConstans.MAX_NUMBER_OF_RECIPES) THEN
	THIS^.uiNumberOfRecipes					:= THIS^.uiNumberOfRecipes + 1;
	THIS^.arrRecipes [THIS^.uiNumberOfRecipes]	:= THIS^.arrRecipes [uiNumberRecipe];
	THIS^.arrRecipes [THIS^.uiNumberOfRecipes].stTexts	:= stTexts;
//	THIS^.arrReceptury [THIS^.uiIloscReceptur].fbNazwa.PowiarzJezyk (fbLokalizacja := THIS^.itfJezyk);	
	AddRecipeFromRecipe				:= TRUE;
END_IF
END_METHOD

(*			
	RafalOS
	Rafał Osajda		03.03.2025		TC 4026.13		wer. 0.0.0.1
	Kopiuje składniki z wybranego szablonu i tworzy nową recepture
*)
METHOD PUBLIC AddRecipeFromTemplate : BOOL
VAR_INPUT
	uiNumberTemplates			: UINT;
	stTexts						: ST_BaseLabel;
END_VAR
IF (THIS^.uiNumberOfRecipes + 1 <= GVL_BaseConstans.MAX_NUMBER_OF_RECIPES) THEN
	THIS^.uiNumberOfRecipes					:= THIS^.uiNumberOfRecipes + 1;
	THIS^.arrRecipes [THIS^.uiNumberOfRecipes]	:= THIS^.arrTemplates [uiNumberTemplates];
	THIS^.arrRecipes [THIS^.uiNumberOfRecipes].stTexts	:= stTexts;
//	THIS^.arrReceptury [THIS^.uiIloscReceptur].fbNazwa.PowiarzJezyk (fbLokalizacja := THIS^.itfJezyk);
	AddRecipeFromTemplate				:= TRUE;
END_IF
END_METHOD

(*			
	RafalOS
	Rafał Osajda		25.10.2025		TC 4024.66
	Dodawanie szablonu - metoda wykorzystywana w zewnętrznym FB tworzenia receptur
*)
METHOD PUBLIC AddTemplate : BOOL
VAR_INPUT
	stTexts			: ST_BaseLabel;
END_VAR
IF (THIS^.uiNumberOfTemplates + 1 <= GVL_BaseConstans.MAX_NUMBER_OF_TEMPLATES) THEN
	THIS^.uiNumberOfTemplates									:= THIS^.uiNumberOfTemplates + 1;
	THIS^.arrTemplates [1].stTexts								:=  stTexts;
	THIS^.arrTemplates [THIS^.uiNumberOfTemplates].uiTemplate	:= THIS^.uiNumberOfTemplates;
	AddTemplate												:= TRUE;
END_IF
END_METHOD

(*			
	RafalOS
	Rafał Osajda		03.03.2025		TC 4026.13		wer. 0.0.0.1
	Przypisuje do referencji wybraną rtecepture
*)
METHOD PUBLIC Choose : BOOL
VAR_INPUT
	uiNumber				: UINT;
END_VAR
//THIS^.refstWybrana				REF= THIS^.arrReceptury [uiNumer];
THIS^.stChosen					:= THIS^.arrRecipes [uiNumber];
THIS^.uiChosen					:= uiNumber;
END_METHOD

(*			
	RafalOS
	Rafał Osajda		25.10.2025		TC 4024.66
	Utworzenie nowych szablonów receptur na podstawie dodanych fb zewnętrznych - wywołanie metody powoduje
	skosowanie dotychczasowych szablonów i receptur
*)
METHOD PUBLIC CreateTemplates : BOOL
VAR_INPUT
END_VAR

VAR
	iI: INT;
END_VAR
THIS^.DeleteRecipes ();
THIS^.DeleteTemplates ();

FOR iI := 1 TO TO_INT (THIS^.uiNumberOfCreatingRecipe) DO
	THIS^.arritfCreatingRecipe [iI].CreateTamplateOfRecipe (itfRecipe := THIS^);
END_FOR
END_METHOD

(*			
	RafalOS
	Rafał Osajda		03.03.2025		TC 4026.13		wer. 0.0.0.1
	
*)
METHOD PUBLIC DeleteRecipe : BOOL
VAR_INPUT
	uiNumber				: uint;
END_VAR
IF (uiNumber > 0 AND uiNumber <= THIS^.uiNumberOfRecipes) THEN

	MEMMOVE (
		destAddr						:= ADR (THIS^.arrRecipes [uiNumber]),
		srcAddr							:= ADR (THIS^.arrRecipes [uiNumber + 1]),
		n								:= SIZEOF (THIS^.arrRecipes [1]) * (GVL_BaseConstans.MAX_NUMBER_OF_RECIPES - (uiNumber))
	);
	THIS^.uiNumberOfRecipes				:= THIS^.uiNumberOfRecipes - 1;
	
	DeleteRecipe			:= TRUE;
END_IF
END_METHOD

(*			
	RafalOS
	Rafał Osajda		30.04.2025		TC 4024.66
	usunięcie wszystkich receptur
*)
METHOD PUBLIC DeleteRecipes : BOOL
VAR_INPUT
END_VAR
MEMSET (
	destAddr			:= ADR (THIS^.arrRecipes),
	fillByte			:= 0,
	n					:= SIZEOF (THIS^.arrRecipes)
);
THIS^.uiNumberOfRecipes 	:= 0;
THIS^.uiChosen			:= 0;
END_METHOD

(*			
	RafalOS
	Rafał Osajda		30.04.2025		TC 4024.66
	usunięcie wszystkich szablonów
*)
METHOD PUBLIC DeleteTemplates : BOOL
VAR_INPUT
END_VAR
MEMSET (
	destAddr			:= ADR (THIS^.arrTemplates),
	fillByte			:= 0,
	n					:= SIZEOF (THIS^.arrTemplates)
);
THIS^.uiNumberOfTemplates 	:= 0;

//THIS^.PowiazJezyk (fbLokalizacja := THIS^.itfJezyk);
END_METHOD

(*			
	RafalOS
	Rafał Osajda		03.03.2025		TC 4026.13		wer. 0.0.0.1
	Zwraca referencje do  receptury
*)
METHOD PUBLIC GetAdressOfRecipe : POINTER TO ST_BaseRecipe
VAR_INPUT
	uiNumber					: UINT;
END_VAR
//IF (__ISVALIDREF (THIS^.refstWybrana )) THEN
//	Zwroc 		:= THIS^.refstWybrana;
//END_IF
GetAdressOfRecipe			:= ADR (THIS^.arrRecipes [uiNumber]);
END_METHOD

(*			
	RafalOS
	Rafał Osajda		03.03.2025		TC 4026.13		wer. 0.0.0.1
	Zwraca referencje do  receptury
*)
METHOD PUBLIC GetChoosen : REFERENCE TO ST_BaseRecipe
//IF (__ISVALIDREF (THIS^.refstWybrana )) THEN
//	Zwroc 		:= THIS^.refstWybrana;
//END_IF
GetChoosen			REF= THIS^.GetReferenceToRecipe (uiNumer := THIS^.uiChosen);
END_METHOD

(*			
	RafalOS
	Rafał Osajda		03.03.2025		TC 4026.13		wer. 0.0.0.1
	
*)
METHOD PUBLIC GetIngredientFromRecipe : ST_BaseDescriptor
VAR_INPUT
	uiNumberOfRecipe			: UINT;
	uiNumberOfIngredient		: UINT;
END_VAR
GetIngredientFromRecipe			:= THIS^.arrRecipes [uiNumberOfRecipe].arrIngredient [uiNumberOfIngredient];
END_METHOD

(*			
	RafalOS
	Rafał Osajda		03.03.2025		TC 4026.13		wer. 0.0.0.1
	
*)
METHOD PUBLIC GetIngredientFromTemplate : ST_BaseDescriptor
VAR_INPUT
	uiNumberOfTemplate			: UINT;
	uiNumberOfIngredient		: UINT;
END_VAR
GetIngredientFromTemplate			:= THIS^.arrRecipes [uiNumberOfTemplate].arrIngredient [uiNumberOfIngredient];
END_METHOD

METHOD PUBLIC GetIsChoosen : BOOL
VAR_INPUT
END_VAR
GetIsChoosen			:= THIS^.uiChosen <> 0;
END_METHOD

METHOD GetNamesOfRecipe : ST_BaseLabel
VAR_INPUT
	uiNumber			: UINT;
END_VAR
GetNamesOfRecipe			:= THIS^.arrRecipes [uiNumber].stTexts;
END_METHOD

METHOD PUBLIC GetNamesOfTemplate : ST_BaseLabel
VAR_INPUT
	uiNumber			: UINT;
END_VAR
GetNamesOfTemplate			:= THIS^.arrTemplates [uiNumber].stTexts;
END_METHOD

(*			
	RafalOS
	Rafał Osajda		03.03.2025		TC 4026.13		wer. 0.0.0.1
	
*)
METHOD PUBLIC GetNumberIngredientOfRecipe : UINT
VAR_INPUT
	uiNumer				: UINT;
END_VAR
GetNumberIngredientOfRecipe 		:= THIS^.arrRecipes [uiNumer].uiNumber;
END_METHOD

METHOD PUBLIC GetNumberIngredientOFTemplate : UINT
VAR_INPUT
	uiNumber				: UINT;
END_VAR
GetNumberIngredientOFTemplate 		:= THIS^.arrTemplates [uiNumber].uiNumber;
END_METHOD

METHOD PUBLIC GetNumberOfChoosen : UINT
VAR_INPUT
END_VAR
GetNumberOfChoosen			:= THIS^.uiChosen;
END_METHOD

METHOD PUBLIC GetNumberOfRecipe : UINT
VAR_INPUT
END_VAR
GetNumberOfRecipe			:= THIS^.uiNumberOfRecipes;
END_METHOD

METHOD PUBLIC GetNumberOfTemplate : UINT
VAR_INPUT
END_VAR
GetNumberOfTemplate		:= THIS^.uiNumberOfTemplates;
END_METHOD

(*			
	RafalOS
	Rafał Osajda		24.03.2025		TC 4024.66
	Zwraca reference do wybranej receptury
*)
METHOD PUBLIC GetReferencesToChoosen : REFERENCE TO ST_BaseRecipe
VAR_INPUT
END_VAR
GetReferencesToChoosen			REF= THIS^.stChosen;
END_METHOD

(*			
	RafalOS
	Rafał Osajda		03.03.2025		TC 4026.13		wer. 0.0.0.1
	Zwraca referencje do  receptury
*)
METHOD PUBLIC GetReferenceToRecipe : REFERENCE TO ST_BaseRecipe
VAR_INPUT
	uiNumer					: UINT;
END_VAR
//IF (__ISVALIDREF (THIS^.refstWybrana )) THEN
//	Zwroc 		:= THIS^.refstWybrana;
//END_IF
GetReferenceToRecipe			REF= THIS^.arrRecipes [uiNumer];
END_METHOD

(*			
	RafalOS
	Rafał Osajda		03.03.2025		TC 4026.13		wer. 0.0.0.1
	Zastępuje wybraną recepture przez istenijącą receputre
*)
METHOD PROTECTED ReplaceRecipeWithAnotherRecipe : BOOL
VAR_INPUT
	uiNumerRecepturyCel			: UINT;
	uiNumerRecepturyZrodlo		: UINT;	
	stNazwa						: ST_BaseLabel;
END_VAR
IF (uiNumerRecepturyCel > 0 AND uiNumerRecepturyCel <= THIS^.uiNumberOfRecipes AND
	uiNumerRecepturyZrodlo > 0 AND uiNumerRecepturyZrodlo <= THIS^.uiNumberOfRecipes AND
	uiNumerRecepturyCel <> uiNumerRecepturyZrodlo) THEN
	THIS^.arrRecipes [uiNumerRecepturyZrodlo]	:= THIS^.arrTemplates [uiNumerRecepturyZrodlo];
	THIS^.arrRecipes [uiNumerRecepturyCel].stTexts	:= stNazwa;
	ReplaceRecipeWithAnotherRecipe 				:= TRUE;
END_IF
END_METHOD

(*			
	RafalOS
	Rafał Osajda		03.03.2025		TC 4026.13		wer. 0.0.0.1
	Zastępuje wybraną recepture przez istenijącą receputre z szablonu
*)
METHOD PUBLIC ReplaceRecipeWithTemplateRecipe : BOOL
VAR_INPUT
	uiNumerRecepturyCel			: UINT;
	uiNumerRecepturyZrodlo		: UINT;
	stNazwa						: ST_BaseLabel;
END_VAR
IF (uiNumerRecepturyCel > 0 AND uiNumerRecepturyCel <= THIS^.uiNumberOfRecipes AND
	uiNumerRecepturyZrodlo > 0 AND uiNumerRecepturyZrodlo <= THIS^.uiNumberOfTemplates) THEN
	THIS^.arrRecipes [uiNumerRecepturyZrodlo]	:= THIS^.arrTemplates [uiNumerRecepturyZrodlo];
	THIS^.arrRecipes [uiNumerRecepturyCel].stTexts	:= stNazwa;
	ReplaceRecipeWithTemplateRecipe 			:= TRUE;
END_IF
END_METHOD

(*			
	RafalOS
	Rafał Osajda		03.06.2025		TC 4024.66
	usuwa referencje do wybranej
*)
METHOD PUBLIC WyczyscWybrana
VAR_INPUT
END_VAR
THIS^.uiChosen := 0;
END_METHOD

(*			
	RafalOS
	Rafał Osajda		16.09.2025		TC 4024.66
	Ustawia numer wybranej receptury na 0 
*)
METHOD PUBLIC WyzerujUstawionaRecepture : BOOL
VAR_INPUT
END_VAR
THIS^.uiChosen			:= 0;
END_METHOD

END_FUNCTION_BLOCK

// ---- POUs/B01_Komunikator/FB_BaseCommunicator.TcPOU
(*			
	RafalOS
	Rafał Osajda		30.07.2025		TC 4024.66
	Głowny fb do kumunikacji pomiędzy fb frameworka
*)
FUNCTION_BLOCK FB_BaseCommunicator IMPLEMENTS ITF_BaseCommunicator
VAR
	arrData					: ARRAY [1..GVL_BaseConstans.MAX_NUMBER_OF_MASSAGES] OF ST_BaseCommunicatorData;
	iNumberOfData			: INT;
	arrStack				: ARRAY [1..GVL_BaseConstans.MAX_NUMBER_OF_MASSAGES_ON_STACK] OF ST_BaseCommunicatorStack;
	iNumberOfitemsInStack	: INT;		//ilość elementów w kolejce
END_VAR

(*			
	RafalOS
	Rafał Osajda		30.07.2025		TC 4024.66
	Dodaje komunikat który będzie wysyłany w systemie. Np. Gotowy wartość TRUE
*)
METHOD PUBLIC AddMessage : INT
VAR_INPUT
	sText				: STRING;
END_VAR
IF (THIS^.iNumberOfData + 1 <= GVL_BaseConstans.MAX_NUMBER_OF_MASSAGES) THEN
	THIS^.iNumberOfData		:= THIS^.iNumberOfData + 1;
	THIS^.arrData [THIS^.iNumberOfData].stMessage.sText		:= sText;
	AddMessage			:= THIS^.iNumberOfData;
ELSE
	AddMessage			:= 0;
END_IF
END_METHOD

METHOD PUBLIC AddRecipientToMessage : BOOL
VAR_INPUT
	iMessageNumber				: INT;
	itfRecipient				: ITF_BaseMessengerRecipient;
END_VAR
IF (THIS^.arrData [iMessageNumber].iNumberOfRecipient + 1 <= GVL_BaseConstans.MAX_NUMBER_OF_CLIENTS) THEN
	THIS^.arrData [iMessageNumber].iNumberOfRecipient			:= THIS^.arrData [iMessageNumber].iNumberOfRecipient + 1;
	THIS^.arrData [iMessageNumber].arritfRecipient [THIS^.arrData [iMessageNumber].iNumberOfRecipient]	:= itfRecipient;
	AddRecipientToMessage									:= TRUE;
END_IF
END_METHOD

METHOD PUBLIC AddSenderToMessage : BOOL
VAR_INPUT
	iMessageNumber		: INT;
	itfSender			: ITF_BaseMessengerSender;
END_VAR
THIS^.arrData [iMessageNumber].itfSender	:= itfSender;
END_METHOD

(*			
	RafalOS
	Rafał Osajda		31.07.2025		TC 4024.66
	
*)
METHOD PRIVATE GetIsMeesageExist : BOOL
VAR_INPUT
	sText			: STRING;
END_VAR
VAR_OUTPUT
	iIndex			: INT;
END_VAR
VAR
	iI				: INT;
END_VAR
FOR iI := 1 TO THIS^.iNumberOfData DO
	IF (sText = THIS^.arrData [iI].stMessage.sText) THEN
		iIndex							:= iI;
		GetIsMeesageExist		:= TRUE;
		RETURN;
	END_IF
END_FOR
GetIsMeesageExist				:= FALSE;
END_METHOD

(*			
	RafalOS
	Rafał Osajda		31.07.2025		TC 4024.66
	Sprawdza czy ten kto nadaje komunikat jest do tego uprawniony
*)
METHOD PRIVATE GetIsRecipientAuthorized : BOOL
VAR_INPUT
	iIndex		: INT;
	itfRecipient	: ITF_BaseMessengerRecipient;
END_VAR
VAR
	iI			: INT;
END_VAR
FOR iI := 1 TO THIS^.arrData [iIndex].iNumberOfRecipient DO
	IF (THIS^.arrData [iIndex].arritfRecipient [iI] = itfRecipient) THEN
		GetIsRecipientAuthorized			:= TRUE;
		RETURN;
	END_IF
END_FOR
GetIsRecipientAuthorized			:= FALSE;
END_METHOD

(*			
	RafalOS
	Rafał Osajda		31.07.2025		TC 4024.66
	Sprawdza czy ten kto nadaje komunikat jest do tego uprawniony
*)
METHOD PRIVATE GetIsSenderAuthorized : BOOL
VAR_INPUT
	iIndex		: INT;
	itfSender	: ITF_BaseMessengerSender;
END_VAR
IF (THIS^.arrData [iIndex].itfSender = itfSender) THEN
	GetIsSenderAuthorized			:= TRUE;
ELSE
	GetIsSenderAuthorized			:= FALSE;
END_IF
END_METHOD

METHOD PUBLIC ReceiveData_BOOL : BOOL
VAR_INPUT
	sText		: STRING;
	itfRecipient	: ITF_BaseMessengerRecipient;
END_VAR
VAR_OUTPUT
	bValue	: BOOL;	
END_VAR
VAR
	iIndex: INT;
END_VAR
IF (THIS^.GetIsMeesageExist (sText := sText, iIndex => iIndex)) THEN
	IF (THIS^.GetIsRecipientAuthorized (iIndex := iIndex, itfRecipient := itfRecipient)) THEN
		bValue				:= THIS^.arrData [iIndex].stMessage.bValue;
		ReceiveData_BOOL			:= TRUE;
		RETURN;
	END_IF
END_IF
ReceiveData_BOOL			:= FALSE;
END_METHOD

METHOD PUBLIC ReceiveData_REAL : BOOL
VAR_INPUT
	sText		: STRING;
	itfRecipient	: ITF_BaseMessengerRecipient;
END_VAR
VAR_OUTPUT
	rValue	: REAL;	
END_VAR
VAR
	iIndex: INT;
END_VAR
IF (THIS^.GetIsMeesageExist (sText := sText, iIndex => iIndex)) THEN
	IF (THIS^.GetIsRecipientAuthorized (iIndex := iIndex, itfRecipient := itfRecipient)) THEN
		rValue				:= THIS^.arrData [iIndex].stMessage.rValue;
		ReceiveData_REAL			:= TRUE;
		RETURN;
	END_IF
END_IF
ReceiveData_REAL			:= FALSE;
END_METHOD

(*			
	RafalOS
	Rafał Osajda		30.07.2025		TC 4024.66
	Wysyła potwierdzenie że odebrał dane
*)
METHOD PUBLIC ReceiveDataConfirm : BOOL
VAR_INPUT
	sText				: STRING;
	itfRecipient			: ITF_BaseMessengerRecipient;
END_VAR
VAR
	iIndex				: INT;
END_VAR
IF (THIS^.GetIsMeesageExist (sText := sText, iIndex => iIndex)) THEN
	IF (THIS^.GetIsRecipientAuthorized (iIndex := iIndex, itfRecipient := itfRecipient)) THEN
		THIS^.iNumberOfitemsInStack		:= THIS^.iNumberOfitemsInStack + 1;
		THIS^.arrStack [THIS^.iNumberOfitemsInStack].stMessage.sText	:= sText;
		THIS^.arrStack [THIS^.iNumberOfitemsInStack].bConfirmation		:= TRUE;
		THIS^.arrStack [THIS^.iNumberOfitemsInStack].itfRecipient			:= itfRecipient;
		ReceiveDataConfirm					:= TRUE;
		RETURN;
	END_IF
END_IF
ReceiveDataConfirm					:= FALSE;
END_METHOD

METHOD SendData_BOOL : BOOL
VAR_INPUT
	sText		: STRING;
	itfSender	: ITF_BaseMessengerSender;
END_VAR
VAR
	iIndex: INT;
END_VAR
IF (THIS^.GetIsMeesageExist (sText := sText, iIndex => iIndex)) THEN
	IF (THIS^.GetIsSenderAuthorized (iIndex := iIndex, itfSender := itfSender)) THEN
		THIS^.iNumberOfitemsInStack	:= THIS^.iNumberOfitemsInStack + 1;
		THIS^.arrStack [THIS^.iNumberOfitemsInStack].stMessage.sText		:= sText;
		THIS^.arrStack [THIS^.iNumberOfitemsInStack].stMessage.bValue		:= TRUE;
		THIS^.arrStack [THIS^.iNumberOfitemsInStack].bSent				:= TRUE;
		SendData_BOOL				:= TRUE;
		RETURN;
	END_IF
END_IF
SendData_BOOL				:= FALSE;
END_METHOD

METHOD SendData_REAL : BOOL
VAR_INPUT
	sText		: STRING;
	rValue		: REAL;
	itfSender	: ITF_BaseMessengerSender;
END_VAR

VAR
	iIndex: INT;
END_VAR
IF (THIS^.GetIsMeesageExist (sText := sText, iIndex => iIndex)) THEN
	IF (THIS^.GetIsSenderAuthorized (iIndex := iIndex, itfSender := itfSender)) THEN
		THIS^.iNumberOfitemsInStack	:= THIS^.iNumberOfitemsInStack + 1;
		THIS^.arrStack [THIS^.iNumberOfitemsInStack].stMessage.sText		:= sText;
		THIS^.arrStack [THIS^.iNumberOfitemsInStack].stMessage.rValue		:= rValue;
		THIS^.arrStack [THIS^.iNumberOfitemsInStack].bSent				:= TRUE;
		SendData_REAL				:= TRUE;
		RETURN;
	END_IF
END_IF
SendData_REAL				:= FALSE;
END_METHOD

METHOD PUBLIC StackSupport
VAR
	iI			: INT;
	iJ			: INT;
	iRecipient	: INT;
	btmpTest	: bool;
END_VAR
IF (iNumberOfitemsInStack > 0) THEN
	FOR iI := 1 TO iNumberOfitemsInStack DO
		IF (THIS^.GetIsMeesageExist (sText := THIS^.arrStack [iI].stMessage.sText, iIndex => iJ)) THEN
			// Nadawanie wiadomosci ustaw odpowiednia wartosc
			IF (THIS^.arrStack [iI].bSent) THEN
				THIS^.arrData [iJ].stMessage.bValue		:= THIS^.arrStack [iI].stMessage.bValue;
				THIS^.arrData [iJ].stMessage.rValue		:= THIS^.arrStack [iI].stMessage.rValue;
				THIS^.arrData [iJ].stMessage.bToPickUp	:= TRUE;
				THIS^.arrData [iJ].iNumberOfConfirmations		:= THIS^.arrData [iJ].iNumberOfRecipient;
			// potwierdzenie odebrania wiadomości wyczyść wiadomość 
			ELSIF (THIS^.arrStack [iI].bConfirmation) THEN
				IF (THIS^.arrData [iJ].iNumberOfRecipient = 1) THEN
					THIS^.arrData [iJ].iNumberOfConfirmations	:= THIS^.arrData [iJ].iNumberOfConfirmations - 1;
					btmpTest		:= TRUE;
				ELSE
					btmpTest		:= TRUE;
					FOR iRecipient := 1 TO THIS^.arrData [iJ].iNumberOfRecipient DO
						IF (THIS^.arrStack [iI].itfRecipient = THIS^.arrData [iJ].arritfRecipient [iRecipient]) THEN
							THIS^.arrData [iJ].arrConfirmations [iRecipient]	:= TRUE;
							THIS^.arrData [iJ].iNumberOfConfirmations			:= THIS^.arrData [iJ].iNumberOfConfirmations - 1;
						END_IF
						btmpTest	:= btmpTest AND THIS^.arrData [iJ].arrConfirmations [iRecipient];
					END_FOR
				END_IF
				IF (btmpTest) THEN
					THIS^.arrData [iJ].stMessage.bToPickUp	:= FALSE;
					THIS^.arrData [iJ].stMessage.bValue		:= FALSE;
					THIS^.arrData [iJ].stMessage.rValue		:= 0;
				END_IF
			END_IF
			EXIT;
		END_IF
	END_FOR
	//wyczyszczenie kolejki
	Tc2_System.MEMSET (
		destAddr			:= ADR (THIS^.arrStack),
		fillByte			:= 0,
		n					:= SIZEOF (THIS^.arrStack)
	);
	THIS^.iNumberOfitemsInStack	:= 0;
END_IF
END_METHOD

END_FUNCTION_BLOCK
